{attribute 'GeneratedUsingTerminal: KL3011'}
{attribute addProperty BoxType "KL3011"}
{attribute addProperty Id "Channel_1AT %Q*Channel_6576A6810"}
{attribute addProperty CRC "1632160004"}
{attribute addProperty Size "0"}
TYPE KL3011_6148C904 :
STRUCT
	{attribute addProperty Name "Channel_1"}
	Channel_1 : Channel_6576A681;
END_STRUCT
END_TYPE

(* stored: Version 1.2.0.0, ProductVersion 3.1.4024.9
   DUT KL3011_6148C904: Id {326b3515-f2fa-47e4-aab1-1478d53e81c8} *)
